PROGRAM _04_Metodo
VAR
	
END_VAR

END_PROGRAM

(* stored: Version 1.1.0.1, ProductVersion 3.1.4024.12
   POU _04_Metodo: Id {0809fefa-bab8-4b56-8e0d-4935fd5424b9}, SpecialFunc None *)
